// Mitsubishi GX Works2 project: PLC 데이터 명령 (INC, DEC, 1씩 증감)   PLC: Q03UDV

PROGRAM MAIN
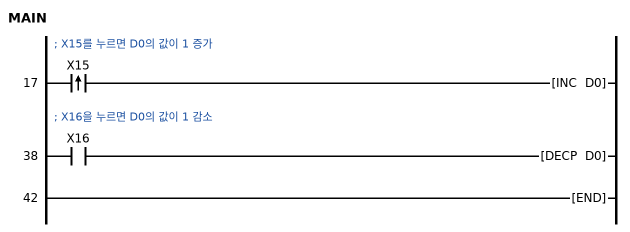
; X15를 누르면 D0의 값이 1 증가
17    LDP     X15
      INC     D0
; X16을 누르면 D0의 값이 1 감소
38    LD      X16
      DECP    D0
42    END
END_PROGRAM
